Staubli VAL3: Day13.dtx

string sInput
lists lResult
  [0]
    string sString
num nResult
num nXcoord
num nYcoord
num nFolds
string sFolds
string sGrid
string sResult
num nFolds_
num nGrid[1 1]
num nLeftMatrix[1 1]
num nRightMatrix[1 1]
num nRowSum
